PROGRAM MAIN
VAR
END_VAR

END_PROGRAM

(* stored: Version 1.1.0.1
   POU MAIN: Id {a49c3faa-87f7-4834-b928-a9efcdb1413e} *)
